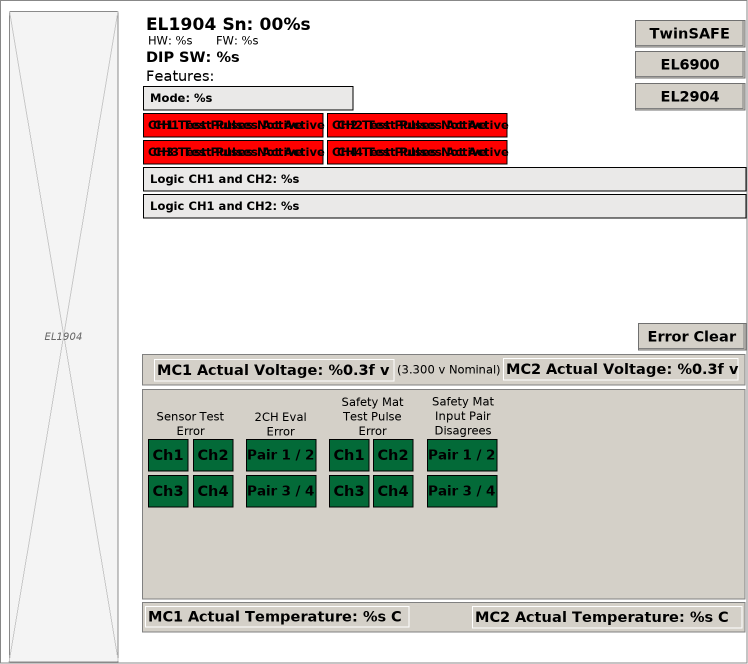
VISUALIZATION EL1904_Specific_Diagnostics  // 748x664
    Button (635,20 110x27), "TwinSAFE"
        OnMouseClick: change screen: TwinSAFE
    Button (635,51 110x27), "EL6900"
        OnMouseClick: change screen: EL6900_Specific_Diagnostics
    Button (635,83 110x27), "EL2904"
        OnMouseClick: change screen: EL2904_Specific_Diagnostics
    Rectangle (143,13 275x22), "EL1904 Sn: 00%s", text variable: g_dwHMI_EL1904Sn
    Rectangle (145,32 65x17), "HW: %s", text variable: g_sHMI_EL1904_HWvers
    Rectangle (213,32 65x17), "FW: %s", text variable: g_sHMI_EL1904_FWvers
    Rectangle (143,46 164x22), "DIP SW: %s", text variable: g_wHMI_EL1904DSw
    Image (9,11 109x651), image: EL1904
    Label (143,65 88x22), "Features:"
    Rectangle (143,86 210x24), "Mode: %s", text variable: g_sHMI_EL1904_OperatingMode
    Button (638,323 108x27), "Error Clear"
        OnMouseUp: execute { g_xHMI_EL1904_ErrClearPB := FALSE ; }
        OnMouseDown: execute { g_xHMI_EL1904_ErrClearPB := TRUE ; }
    Group (142,354 603x31)
        Rectangle (0,0 603x31)
        Label (251,8 112x15), "(3.300 v Nominal)"
        Rectangle (12,5 240x22), "MC1 Actual Voltage: %0.3f v", text variable: g_wHMI_EL1904PriMC_Volts
        Rectangle (361,4 235x22), "MC2 Actual Voltage: %0.3f v", text variable: g_wHMI_EL1904SecMC_Volts
    Group (142,602 603x30)
        Rectangle (0,0 603x30)
        Rectangle (3,4 264x21), "MC1 Actual Temperature: %s C", text variable: g_wHMI_EL1904PriMCTemp
        Rectangle (330,4 270x22), "MC2 Actual Temperature: %s C", text variable: g_wHMI_EL1904SecMCTemp
    Rectangle (142,389 603x210)
    Label (151,408 79x32), "Sensor Test Error"
    Rectangle (148,439 40x32), "Ch1", colour toggle: g_xHMI_EL1904SenT1
    Rectangle (193,439 40x32), "Ch2", colour toggle: g_xHMI_EL1904SenT2
    Rectangle (148,475 40x32), "Ch3", colour toggle: g_xHMI_EL1904SenT3
    Rectangle (193,475 40x32), "Ch4", colour toggle: g_xHMI_EL1904SenT4
    Label (331,389 83x55), "Safety Mat Test Pulse Error"
    Rectangle (329,439 40x32), "Ch1", colour toggle: g_xHMI_EL1904_SMExtSupply_CH1
    Rectangle (373,439 40x32), "Ch2", colour toggle: g_xHMI_EL1904_SMExtSupply_CH2
    Rectangle (329,475 40x32), "Ch3", colour toggle: g_xHMI_EL1904_SMExtSupply_CH3
    Rectangle (373,475 40x32), "Ch4", colour toggle: g_xHMI_EL1904_SMExtSupply_CH4
    Rectangle (246,439 70x32), "Pair 1 / 2", colour toggle: g_xHMI_EL1904_2CHEval_Pair1
    Rectangle (246,475 70x32), "Pair 3 / 4", colour toggle: g_xHMI_EL1904_2CHEval_Pair2
    Label (247,408 67x33), "2CH Eval Error"
    Rectangle (427,439 70x32), "Pair 1 / 2", colour toggle: g_xHMI_EL1904_SMiPair_Pair1
    Rectangle (427,475 70x32), "Pair 3 / 4", colour toggle: g_xHMI_EL1904_SMiPair_Pair2
    Label (419,392 88x48), "Safety Mat Input Pair Disagrees"
    Rectangle (143,167 603x24), "Logic CH1 and CH2: %s", text variable: g_sHMI_EL1904_LogicCh1andCh2
    Rectangle (143,194 603x24), "Logic CH1 and CH2: %s", text variable: g_sHMI_EL1904_LogicCh3andCh4
    Rectangle (327,113 180x24), colour toggle: g_xHMI_EL1904_SensTestActive2
    Rectangle (143,113 180x24), colour toggle: g_xHMI_EL1904_SensTestActive1
    Rectangle (327,140 180x24), colour toggle: g_xHMI_EL1904_SensTestActive4
    Rectangle (143,140 180x24), colour toggle: g_xHMI_EL1904_SensTestActive3
    Group (145,110 177x30)
        Label (5,0 167x30), "CH1 Test Pulses Active", invisible if: NOT g_xHMI_EL1904_SensTestActive1
        Label (0,0 177x30), "CH1 Test Pulses Not Active", invisible if: g_xHMI_EL1904_SensTestActive1
    Group (329,110 177x30)
        Label (5,0 167x30), "CH2 Test Pulses Active", invisible if: NOT g_xHMI_EL1904_SensTestActive2
        Label (0,0 177x30), "CH2 Test Pulses Not Active", invisible if: g_xHMI_EL1904_SensTestActive2
    Group (145,137 177x30)
        Label (5,0 167x30), "CH3 Test Pulses Active", invisible if: NOT g_xHMI_EL1904_SensTestActive3
        Label (0,0 177x30), "CH3 Test Pulses Not Active", invisible if: g_xHMI_EL1904_SensTestActive3
    Group (329,137 177x30)
        Label (5,0 167x30), "CH4 Test Pulses Active", invisible if: NOT g_xHMI_EL1904_SensTestActive4
        Label (0,0 177x30), "CH4 Test Pulses Not Active", invisible if: g_xHMI_EL1904_SensTestActive4
END_VISUALIZATION

(* stored: Version 1.1.0.1, ProductVersion 3.1.0.18
   Visu EL1904_Specific_Diagnostics: Id {c787502f-95ff-47cb-8021-79a9dc3784a4} *)
